PROGRAM MAIN
VAR
END_VAR

Kuka();

END_PROGRAM

(* stored: Version 1.1.0.1, ProductVersion 3.1.4024.12
   POU MAIN: Id {093faa6d-62d8-4703-ba60-8d584e27ea50}, SpecialFunc None *)
